# EPICS autosave request: automation1App/Db/Automation1ProfileMoveController_settings.req
$(P)$(R)PulseMode
$(P)$(R)PulseDir
$(P)$(R)PulseLength
$(P)$(R)PulsePeriod
$(P)$(R)PulseSrc
$(P)$(R)PulseOut
$(P)$(R)PulseAxis
$(P)$(R)NumPulsePositions
